FUNCTION_BLOCK FB_02_BuidGroup

VAR_INPUT
	bExecute:BOOL;
	nXAxisId:UDINT;
	nYAxisId:UDINT;
	nZAxisId:UDINT;
	nQ1AxisId:UDINT;
	nQ2AxisId:UDINT;
END_VAR
VAR_OUTPUT
	bBusy:BOOL;(*功能块执行忙标志*)
	bError:BOOL;(*出错*)
	bDone:BOOL;(*执行完毕*)
END_VAR
VAR_IN_OUT
//	stX:AXIS_REF;
//	stY:AXIS_REF;
//	stZ:AXIS_REF;
	stItpToPlc :NCTOPLC_NCICHANNEL_REF;
	stPlcToItp:PLCTONC_NCICHANNEL_REF;
END_VAR
VAR
	BuidGroupStep:INT:=0;
	fbBuidGroup:CfgBuildExt3DGroup;(*配置NciGroup*)
END_VAR

CASE BuidGroupStep OF
	0:
	  IF  bExecute THEN
		 bBusy:=TRUE;(*FB执行状态*)
		  bDone:=FALSE;(*FB执行完毕*)
		  bError:=FALSE;(*报错*)
		  BuidGroupStep:=10;(*进入10步*) 
	  END_IF
	10:
	  fbBuidGroup(
	    bExecute:= TRUE, 
	    nGroupId:= ItpGetGroupId(sNciToPlc:=stItpToPlc), 
	    nXAxisId:= nXAxisId, 
	    nYAxisId:= nYAxisId, 
	    nZAxisId:= nZAxisId, 
	    nQ1AxisId:= nQ1AxisId, 
	    nQ2AxisId:= nQ2AxisId, 
	    nQ3AxisId:= 0, 
	    nQ4AxisId:= 0, 
	    nQ5AxisId:= 0, 
	    tTimeOut:= , 
	    bBusy=> , 
	    bErr=> , 
	    nErrId=> );
	   IF NOT fbBuidGroup.bBusy THEN
		  IF NOT fbBuidGroup.bErr THEN
			BuidGroupStep:=20;(*进入20步*)  
		  ELSE
			bBusy:=FALSE;
			bError:=TRUE;
			BuidGroupStep:=999;
		  END_IF
		fbBuidGroup(bExecute:= FALSE,nGroupId:= ItpGetGroupId(sNciToPlc:=stItpToPlc));
	    END_IF
	 20:
	   //ItpSetOverridePercent(fOverridePercent:= 100, sPlcToNci:= stPlcToItp);
	   bDone:=TRUE;
       bBusy:=FALSE;   
	   IF NOT bExecute THEN
		 BuidGroupStep:=0;
	   END_IF
	 999:
	   IF NOT bExecute THEN		   
	    BuidGroupStep:=0;
        bError:=FALSE; 
	 END_IF
END_CASE

END_FUNCTION_BLOCK

(* stored: Version 1.1.0.1, ProductVersion 3.1.4024.12
   POU FB_02_BuidGroup: Id {c2a71bfc-09e9-4bf9-b476-9c80c5c9d727}, SpecialFunc None *)
